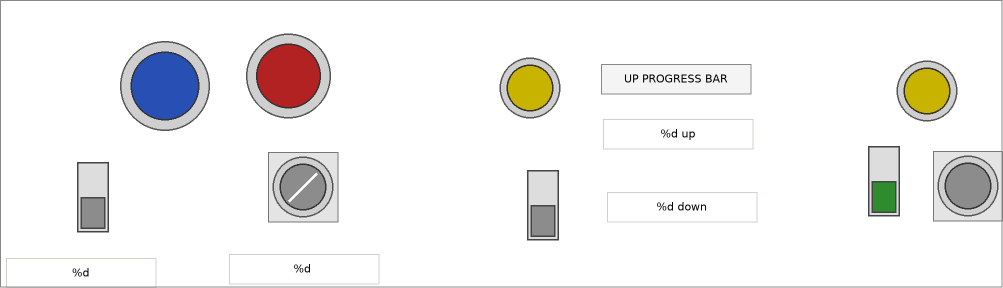
VISUALIZATION Visualization  // 1003x288
    DipSwitch (58,162 70x70), variable: GVL.S1, behaviour: TOGGLE, style: Switch-DipSwitch-Gray
    RotarySwitch (268,152 70x70), variable: GVL.S2, behaviour: TOGGLE, style: Switch-RotarySwitch-Gray
    Lamp1 (113,33 104x106), variable: GVL.LED1, invisible if: GVL.S3, style: Lamp-Lamp1-Blue
    Textfield (6,258 150x30), "%d", text variable: GVL.counter
        OnDialogClosed: write the text variable via Default
    Textfield (229,254 150x30), "%d", text variable: MAIN1.counter1
        OnDialogClosed: write the text variable via Edit
    Lamp1 (495,53 70x70), variable: GVL.flasher, style: Lamp-Lamp1-Yellow
    DipSwitch (508,170 70x70), tooltip "%S", variable: GVL.S3, behaviour: TOGGLE, style: Switch-DipSwitch-Gray
    Textfield (603,119 150x30), "%d up", text variable: MAIN1.edge
    Textfield (607,192 150x30), "%d down", text variable: MAIN1.FALL
    DipSwitch (849,146 70x70), tooltip "reset", variable: GVL.S4, behaviour: TOGGLE, style: Switch-DipSwitch-Green
    PushSwitch (933,151 70x70), variable: GVL.S4, behaviour: TAP, style: Switch-PushSwitch-Gray
    Progressbar (601,64 150x30), "UP PROGRESS BAR", variable: MAIN1.edge, invisible if: MAIN1.edge>50
    Lamp1 (239,27 99x98), variable: GVL.LED2, invisible if: GVL.LED1, style: Lamp-Lamp1-Red
    Lamp1 (892,56 70x70), variable: GVL.LED4, style: Lamp-Lamp1-Yellow
END_VISUALIZATION

(* stored: Version 1.1.0.1, ProductVersion 3.1.4024.12
   Visu Visualization: Id {dd173a1b-fe87-4c90-9ecd-275ff47a3dd1} *)
